TYPE ref_upperLower :
STRUCT
	upperLower : ARRAY[1..2] OF ref_cav ;
END_STRUCT
END_TYPE

(* stored: Version 1.1.0.1, ProductVersion 3.1.4024.11
   DUT ref_upperLower: Id {8e070547-316d-4358-be46-fcf60ea7a436} *)
